Universal Robots PolyScope program: tcp0test.urp

Program tcp0test (installation=default directory=/home/ros/ursim-5.13.0.113898/programs createdIn=5.13.0 lastSavedIn=5.13.0 robotSerialNumber=20195299999)
Calibrated DH parameters: a=[0, -0.6127, -0.57155, 0, 0, 0]; d=[0.1807, 0, 0, 0.17415, 0.11985, 0.11655]; alpha=[1.570796, 0, 0, 1.570796, -1.570796, 0]; deltaTheta=[0, 0, 0, 0, 0, 0]
InitVariablesNode
Robot Program (runOnlyOnce=false)
  Placeholder
